// TIA Portal V18 export
DATA_BLOCK "_hmi_spot_manager_DB"   // DB51
VERSION : 0.1
// stored: AutoNumber true, DBAccessibleFromOPCUA true, InstanceOfName _hmi_spot_manager, InstanceOfType FB
"_hmi_spot_manager"
   // VAR_INPUT
   //    cur_pos_set : "typePositions";
   // END_VAR
   // VAR_OUTPUT
   //    hmi_pos_set : "typePositions";
   //    hmi_to_spot_allowed : Bool;
   //    Spot_positions_now : "typePositions";
   // END_VAR
   // VAR_IN_OUT
   //    spot_set_encoder : Bool;
   //    spot_set_hmi : Bool;
   // END_VAR
   // VAR
   //    spot_ws : WString;
   //    part_was : Int;
   //    spotSaver { S7_SetPoint := 'True'} : "_hmi_singleSpotManager";
   // END_VAR
BEGIN
END_DATA_BLOCK
